(* CoDeSys 2.3.9.37 project: Cap6_2.pro *)
(* Libraries: Standard.lib 4.10.05 12:14:46 *)

(* POU PLC_PRG, LD *)
PROGRAM PLC_PRG
VAR
    (* Entradas *)
	A: BOOL;
       B:BOOL;
    (* Salidas *)
   	S1: BOOL;
      S2 :BOOL;
    (* Instancias de bloques funcionales *)
	DetectorBajada: F_TRIG;
END_VAR
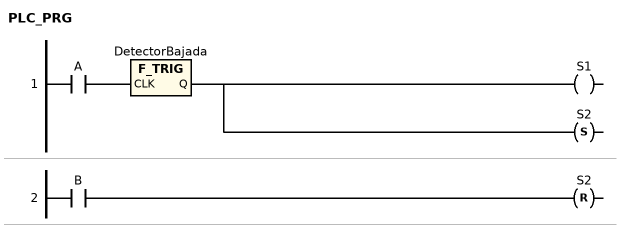
_LD_ (* Ladder Diagram *)
NETWORK 1
	[A] - DetectorBajada:F_TRIG(CLK: *) --- (S1) (S S2)
NETWORK 2
	[B] --- (R S2)
_END_LD_
(* the same logic as Structured Text *)
(* Network 1 *)
DetectorBajada(CLK := A);
S1 := DetectorBajada.Q;
IF DetectorBajada.Q THEN S2 := TRUE; END_IF;
(* Network 2 *)
IF B THEN S2 := FALSE; END_IF;
END_PROGRAM

(* Visualisation Visu
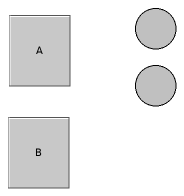
button at (42,51)-(103,122): text "A"; taps PLC_PRG.A
ellipse at (168,44)-(209,85): alarm colour if PLC_PRG.S1
ellipse at (168,101)-(209,142): alarm colour if PLC_PRG.S2
button at (41,153)-(102,224): text "B"; taps PLC_PRG.B
2 elements of other kinds (tables, trends, ...) not read
*)
